// Mitsubishi GX Works2 project: 0625(카운트)   PLC: Q02/Q02H

PROGRAM MAIN
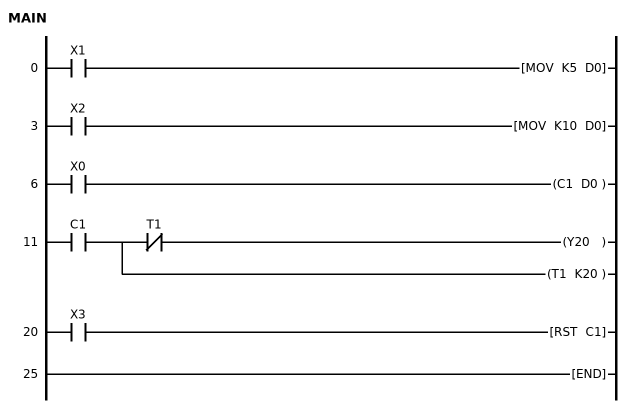
0     LD      X1
      MOV     K5 D0
3     LD      X2
      MOV     K10 D0
6     LD      X0
      OUT     C1 D0
11    LD      C1
      MPS
      ANI     T1
      OUT     Y20
      MPP
      OUT     T1 K20
20    LD      X3
      RST     C1
25    END
END_PROGRAM
